// TIA Portal V17 export
// export: Created 2022-12-08T10:20:57.686031Z, ExportSetting WithDefaults, DisplayName Totally Integrated Automation Portal, DisplayVersion V17 Update 5, DisplayName TIA Portal Openness, DisplayVersion V17 Update 5, DisplayName TIA Portal Version Control Interface, DisplayVersion V17, DisplayName Simotion SCOUT TIA, DisplayVersion 5.4.3.0, DisplayName SINAMICS Startdrive Advanced, DisplayVersion V17 SP1, DisplayName SINAMICS Startdrive G130, G150, S120, S150, SINAMICS MV, S210, DisplayVersion V17 SP1, DisplayName SINAMICS Startdrive G110M, G120, G120C, G120D, G120P, G115D, DisplayVersion V17 SP1, DisplayName STEP 7 Professional, DisplayVersion V17 Update 5, DisplayName STEP 7 Safety, DisplayVersion V17, DisplayName WinCC Advanced, DisplayVersion V17 Update 5
FUNCTION_BLOCK "FB_GearInWithOffset"   // FB1311, FBD
TITLE = Gleichlauf mit Offset
{ S7_Optimized_Access := 'TRUE' }
VERSION : 0.1
// stored: AutoNumber false, IsIECCheckEnabled true, IsRetainMemResEnabled false, MemoryReserve 100, SetENOAutomatically true, UDAEnableTagReadback false
   VAR_INPUT
      Master { ExternalAccessible := 'False'; ExternalVisible := 'False'; ExternalWritable := 'False'} : DB_ANY;
      Slave { ExternalAccessible := 'False'; ExternalVisible := 'False'; ExternalWritable := 'False'} : DB_ANY;
      Offset_Plus : Bool;
      Offset_Minus : Bool;
      "Einkoppeln ohne Bewegung" : Bool;
      Start : Bool;
      Richtung : Int := 1;   // 1 - Positiv, 2 - Negativ, 3 - kürzester Weg
      Velocity : LReal := -1.0;   // Geschwindigkeit
      Acceleration : LReal := -1.0;   // Beschleunigung
      Deceleration : LReal := -1.0;   // Verzögerung
      Jerk : LReal := -1.0;   // Ruck
      RatioNumerator : LReal := 1.0;
      RatioDenominator : LReal := 1.0;
   END_VAR
   VAR_OUTPUT
      InGear : Bool;
      Error : Bool;
      ErrorID : Word;
   END_VAR
   VAR_IN_OUT
      AchsData : "UDT_ServoData";
   END_VAR
   VAR
      Flanken : Struct
         "Fp Plus" : Bool;
         "Fp Minus" : Bool;
      END_STRUCT;
      MoveAbsolut { S7_SetPoint := 'True'} : "LAnyAxis_MC_MoveAbsolute";
      GearIn { S7_SetPoint := 'True'} : "LAnyAxis_MC_GearIn";
      PhasingRelativ { S7_SetPoint := 'True'} : "LAnyAxis_MC_PhasingRelative";
      ActualData_Slave { S7_SetPoint := 'True'} : "UDT_ServoActualData";
      ActualData_Master { S7_SetPoint := 'True'} : "UDT_ServoActualData";
      l_Offset_alt { S7_SetPoint := 'True'} : LReal;
      l_Offset_pos { S7_SetPoint := 'True'} : LReal;
      l_Verschiebung : LReal;
      l_PosMove : LReal;
      l_Offsetänderung : LReal;
      l_ErrorID : Word;
      StartPhasing : Bool;
      l_Numerator : LReal;
      l_Denominator : LReal;
      l_Getriebeänderung : Bool;
      word_ret_val : Word;
   END_VAR
   VAR_TEMP   // added for the SCL form of the ladder/FBD networks
      _w1 : Bool;
      _w2 : Bool;
   END_VAR
BEGIN

REGION Network 1: ActualData lesen
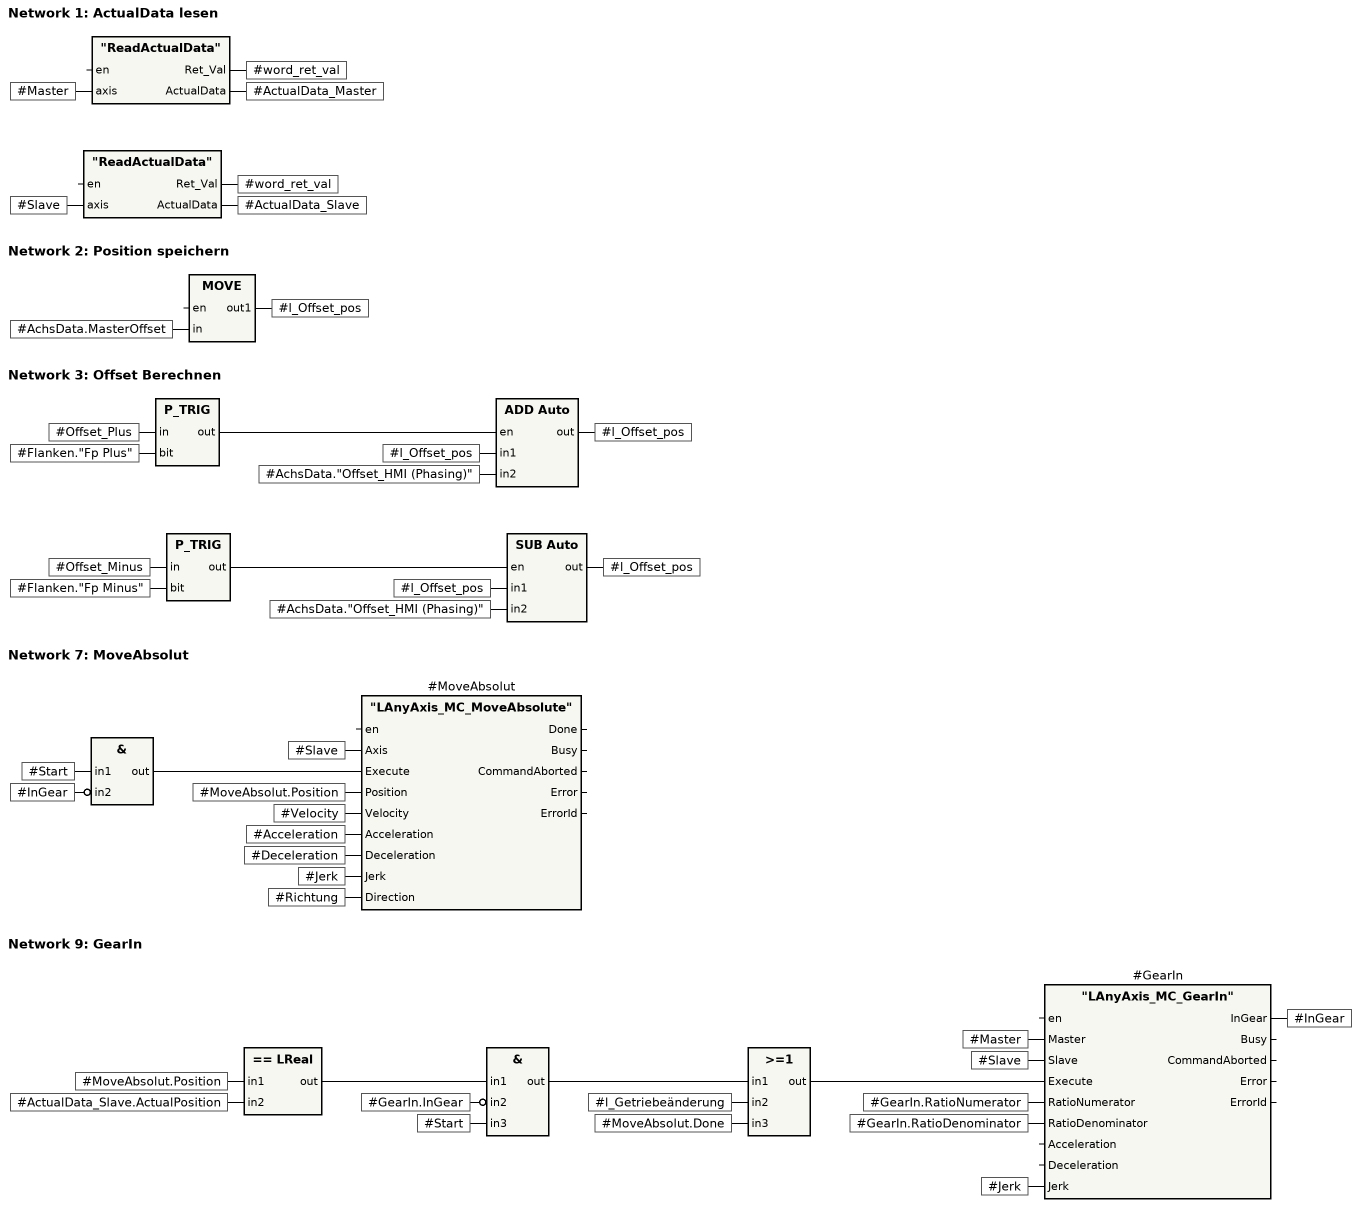
   #word_ret_val := "ReadActualData"(axis := #Master, ActualData => #ActualData_Master);
   #word_ret_val := "ReadActualData"(axis := #Slave, ActualData => #ActualData_Slave);
END_REGION

REGION Network 2: Position speichern
   #l_Offset_pos := #AchsData.MasterOffset;
END_REGION

REGION Network 3: Offset Berechnen
   #_w1 := #Offset_Plus AND NOT #Flanken."Fp Plus";   // rising edge
   #Flanken."Fp Plus" := #Offset_Plus;
   IF #_w1 THEN #l_Offset_pos := #l_Offset_pos + #AchsData."Offset_HMI (Phasing)"; END_IF;
   #_w2 := #Offset_Minus AND NOT #Flanken."Fp Minus";   // rising edge
   #Flanken."Fp Minus" := #Offset_Minus;
   IF #_w2 THEN #l_Offset_pos := #l_Offset_pos - #AchsData."Offset_HMI (Phasing)"; END_IF;
END_REGION

REGION Network 4 (SCL): Offsetberechnung
   IF NOT #InGear THEN
       IF #l_Offset_pos >= #ActualData_Slave.Modulo THEN
           #l_Offset_pos := #l_Offset_pos - #ActualData_Slave.Modulo;
       END_IF;

       IF #l_Offset_pos < 0 THEN
           #l_Offset_pos := #ActualData_Slave.Modulo + #l_Offset_pos;
       END_IF;
       #l_Offset_alt := #l_Offset_pos;
   END_IF;
END_REGION

REGION Network 5 (SCL): Offsetänderung berechnung
   IF #InGear
       AND #l_Offset_pos <> #l_Offset_alt
       AND NOT #StartPhasing
   THEN
       #l_Offsetänderung := #l_Offset_pos - #l_Offset_alt;
       #l_Offset_alt := #l_Offset_pos;
       #StartPhasing := true;
   END_IF;
END_REGION

REGION Network 6 (SCL): Position berechnen
   IF #l_Offset_pos >= #ActualData_Slave.Modulo / 2 THEN
       #l_Verschiebung := #l_Offset_pos - #ActualData_Slave.Modulo;
   ELSE
       #l_Verschiebung := (#l_Offset_pos+#ActualData_Slave.Modulo) - #ActualData_Slave.Modulo;
   END_IF;

   IF NOT #"Einkoppeln ohne Bewegung"
   THEN
       #MoveAbsolut.Position := ((#ActualData_Slave.Modulo / #ActualData_Master.Modulo) * #ActualData_Master.ActualPosition) + #l_Verschiebung;
   ELSE
       #MoveAbsolut.Position := #ActualData_Slave.ActualPosition;
   END_IF;
END_REGION

REGION Network 7: MoveAbsolut
   #MoveAbsolut(Axis := #Slave,   // "LAnyAxis_MC_MoveAbsolute"
                Execute := #Start AND NOT #InGear,
                Position := #MoveAbsolut.Position,
                Velocity := #Velocity,
                Acceleration := #Acceleration,
                Deceleration := #Deceleration,
                Jerk := #Jerk,
                Direction := #Richtung);
END_REGION

REGION Network 8 (SCL): Ratio Numerator und Ratio Denominator umrechnen
   IF NOT #GearIn.InGear
   THEN
       #l_Numerator := #RatioNumerator;
       #l_Denominator := #RatioDenominator;
   END_IF;

   IF #GearIn.InGear
       AND (#l_Numerator <> #RatioNumerator
       OR #l_Denominator <> #RatioDenominator)
   THEN
       #l_Numerator := #RatioNumerator;
       #l_Denominator := #RatioDenominator;
       #l_Getriebeänderung := true;
   END_IF;

   #GearIn.RatioNumerator := LREAL_TO_DINT(#l_Numerator);

   //Wenn Numerator <= 0 wird dieser auf den Wert des Denominator gesetz um die Null zu vermeiden
   IF #RatioNumerator <= 0.0
   THEN
       #GearIn.RatioNumerator := LREAL_TO_DINT(#l_Denominator);
   END_IF;

   #GearIn.RatioDenominator := LREAL_TO_DINT(#l_Denominator);
END_REGION

REGION Network 9: GearIn
   // #Acceleration
   // #Deceleration
   #GearIn(Master := #Master,   // "LAnyAxis_MC_GearIn"
           Slave := #Slave,
           Execute := ((#MoveAbsolut.Position = #ActualData_Slave.ActualPosition) AND NOT #GearIn.InGear AND #Start) OR #l_Getriebeänderung OR #MoveAbsolut.Done,
           RatioNumerator := #GearIn.RatioNumerator,
           RatioDenominator := #GearIn.RatioDenominator,
           Jerk := #Jerk,
           InGear => #InGear);
END_REGION

REGION Network 10 (SCL): Getriebeänderung zurücksetzen
   IF #GearIn.InGear
       AND #l_Numerator = #RatioNumerator
       AND #l_Denominator = #RatioDenominator
   THEN
       #l_Getriebeänderung := false;
   END_IF;
END_REGION

REGION Network 11: Phasing
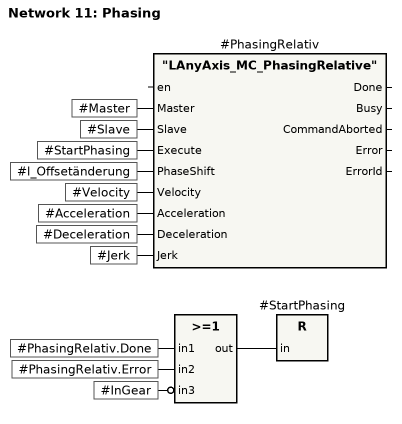
   #PhasingRelativ(Master := #Master,   // "LAnyAxis_MC_PhasingRelative"
                   Slave := #Slave,
                   Execute := #StartPhasing,
                   PhaseShift := #l_Offsetänderung,
                   Velocity := #Velocity,
                   Acceleration := #Acceleration,
                   Deceleration := #Deceleration,
                   Jerk := #Jerk);
   IF #PhasingRelativ.Done OR #PhasingRelativ.Error OR NOT #InGear THEN #StartPhasing := FALSE; END_IF;
END_REGION

REGION Network 12 (SCL): aktuelle Verschiebung
   IF #InGear THEN
       IF #l_Offset_pos >= #ActualData_Master.Modulo THEN
           #l_Offset_pos := #l_Offset_pos - #ActualData_Master.Modulo;
       END_IF;

       IF #l_Offset_pos < 0 THEN
           #l_Offset_pos := #ActualData_Master.Modulo + #l_Offset_pos;
       END_IF;
   END_IF;

   #AchsData.MasterOffset := #l_Offset_pos;
END_REGION

REGION Network 13 (SCL): Error
   #Error := #MoveAbsolut.Error OR #GearIn.Error;

   #l_ErrorID := 16#0000;

   IF #MoveAbsolut.Error THEN
       #l_ErrorID := #MoveAbsolut.ErrorId;
   END_IF;

   IF #GearIn.Error THEN
       #l_ErrorID := #GearIn.ErrorId;
   END_IF;

   #ErrorID := #l_ErrorID;
END_REGION
END_FUNCTION_BLOCK
